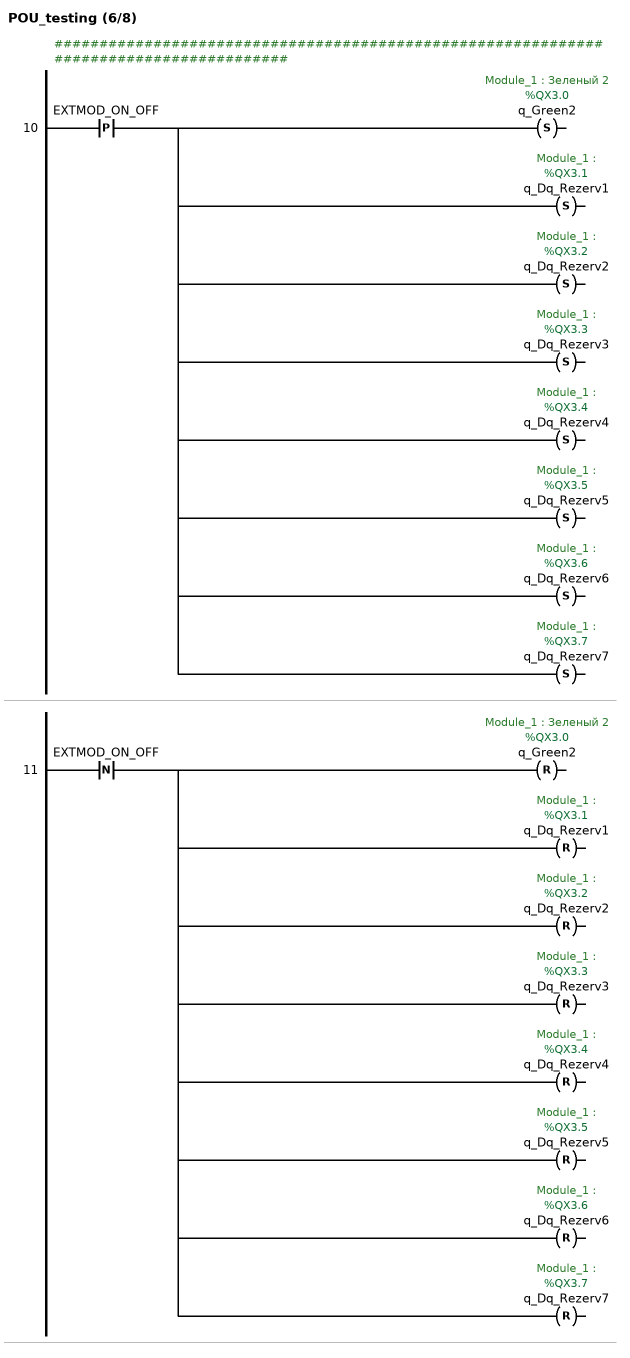
// NETWORK 10
// #######################################################################################
//   q_Green2: Module_1 : Зеленый 2 | AT %QX3.0
//   q_Dq_Rezerv1: Module_1 : | AT %QX3.1
//   q_Dq_Rezerv2: Module_1 : | AT %QX3.2
//   q_Dq_Rezerv3: Module_1 : | AT %QX3.3
//   q_Dq_Rezerv4: Module_1 : | AT %QX3.4
//   q_Dq_Rezerv5: Module_1 : | AT %QX3.5
//   q_Dq_Rezerv6: Module_1 : | AT %QX3.6
//   q_Dq_Rezerv7: Module_1 : | AT %QX3.7
_rt5(CLK := EXTMOD_ON_OFF);
q_Green2 S= _rt5.Q;
q_Dq_Rezerv1 S= _rt5.Q;
q_Dq_Rezerv2 S= _rt5.Q;
q_Dq_Rezerv3 S= _rt5.Q;
q_Dq_Rezerv4 S= _rt5.Q;
q_Dq_Rezerv5 S= _rt5.Q;
q_Dq_Rezerv6 S= _rt5.Q;
q_Dq_Rezerv7 S= _rt5.Q;

// NETWORK 11
//   q_Green2: Module_1 : Зеленый 2 | AT %QX3.0
//   q_Dq_Rezerv1: Module_1 : | AT %QX3.1
//   q_Dq_Rezerv2: Module_1 : | AT %QX3.2
//   q_Dq_Rezerv3: Module_1 : | AT %QX3.3
//   q_Dq_Rezerv4: Module_1 : | AT %QX3.4
//   q_Dq_Rezerv5: Module_1 : | AT %QX3.5
//   q_Dq_Rezerv6: Module_1 : | AT %QX3.6
//   q_Dq_Rezerv7: Module_1 : | AT %QX3.7
_ft3(CLK := EXTMOD_ON_OFF);
q_Green2 R= _ft3.Q;
q_Dq_Rezerv1 R= _ft3.Q;
q_Dq_Rezerv2 R= _ft3.Q;
q_Dq_Rezerv3 R= _ft3.Q;
q_Dq_Rezerv4 R= _ft3.Q;
q_Dq_Rezerv5 R= _ft3.Q;
q_Dq_Rezerv6 R= _ft3.Q;
q_Dq_Rezerv7 R= _ft3.Q;

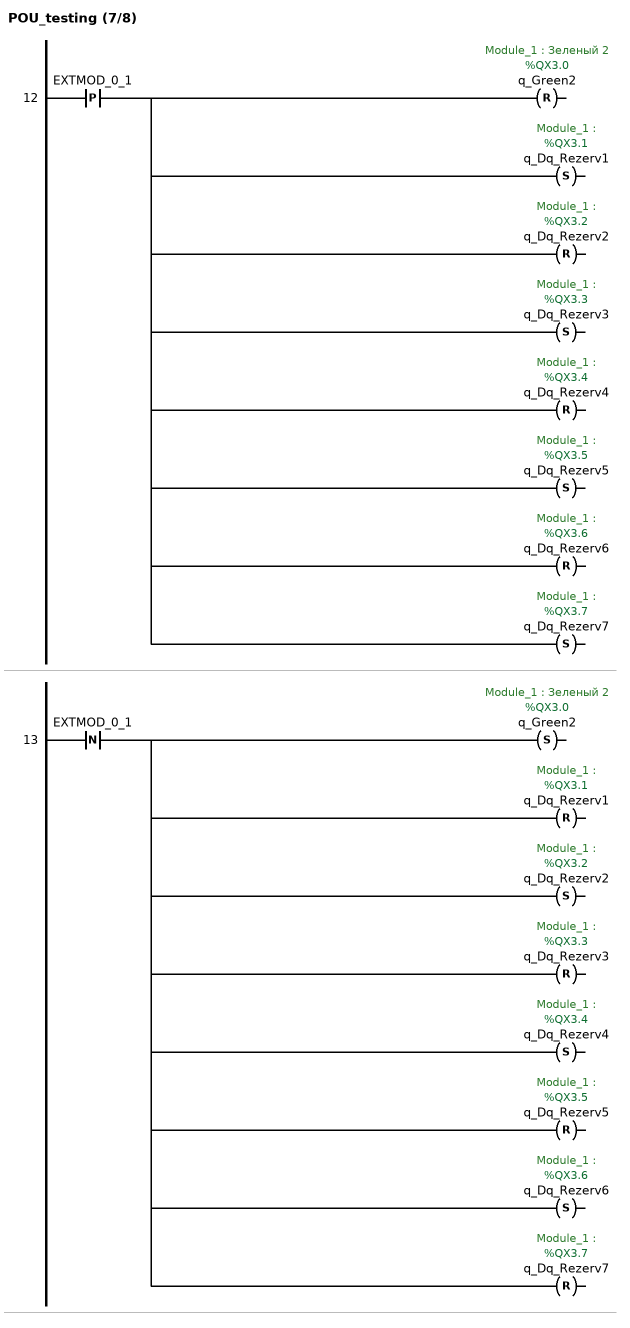
// NETWORK 12
//   q_Green2: Module_1 : Зеленый 2 | AT %QX3.0
//   q_Dq_Rezerv1: Module_1 : | AT %QX3.1
//   q_Dq_Rezerv2: Module_1 : | AT %QX3.2
//   q_Dq_Rezerv3: Module_1 : | AT %QX3.3
//   q_Dq_Rezerv4: Module_1 : | AT %QX3.4
//   q_Dq_Rezerv5: Module_1 : | AT %QX3.5
//   q_Dq_Rezerv6: Module_1 : | AT %QX3.6
//   q_Dq_Rezerv7: Module_1 : | AT %QX3.7
_rt6(CLK := EXTMOD_0_1);
q_Green2 R= _rt6.Q;
q_Dq_Rezerv1 S= _rt6.Q;
q_Dq_Rezerv2 R= _rt6.Q;
q_Dq_Rezerv3 S= _rt6.Q;
q_Dq_Rezerv4 R= _rt6.Q;
q_Dq_Rezerv5 S= _rt6.Q;
q_Dq_Rezerv6 R= _rt6.Q;
q_Dq_Rezerv7 S= _rt6.Q;

// NETWORK 13
//   q_Green2: Module_1 : Зеленый 2 | AT %QX3.0
//   q_Dq_Rezerv1: Module_1 : | AT %QX3.1
//   q_Dq_Rezerv2: Module_1 : | AT %QX3.2
//   q_Dq_Rezerv3: Module_1 : | AT %QX3.3
//   q_Dq_Rezerv4: Module_1 : | AT %QX3.4
//   q_Dq_Rezerv5: Module_1 : | AT %QX3.5
//   q_Dq_Rezerv6: Module_1 : | AT %QX3.6
//   q_Dq_Rezerv7: Module_1 : | AT %QX3.7
_ft4(CLK := EXTMOD_0_1);
q_Green2 S= _ft4.Q;
q_Dq_Rezerv1 R= _ft4.Q;
q_Dq_Rezerv2 S= _ft4.Q;
q_Dq_Rezerv3 R= _ft4.Q;
q_Dq_Rezerv4 S= _ft4.Q;
q_Dq_Rezerv5 R= _ft4.Q;
q_Dq_Rezerv6 S= _ft4.Q;
q_Dq_Rezerv7 R= _ft4.Q;

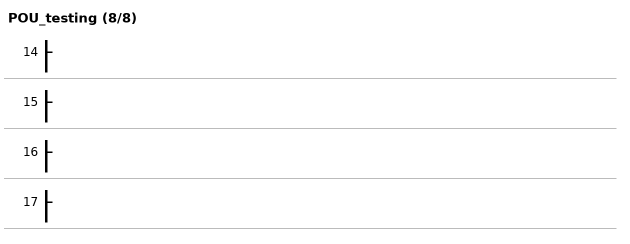
// NETWORK 14

// NETWORK 15

// NETWORK 16

// NETWORK 17

END_PROGRAM

// MyController/Application/POU_testing_modbus
PROGRAM POU_testing_modbus

VAR
	button_light AT %MW1001: BOOL;
END_VAR

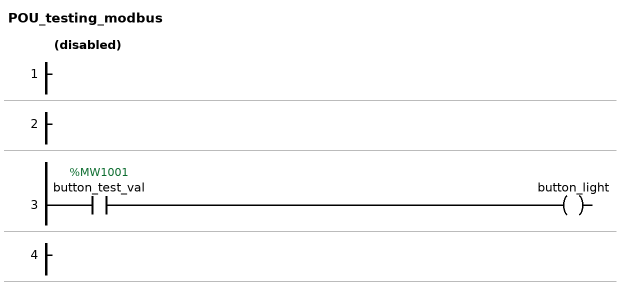
// NETWORK 1 (disabled)

// NETWORK 2

// NETWORK 3
//   button_test_val: AT %MW1001
button_light := button_test_val;

// NETWORK 4

END_PROGRAM
